INTERFACE I_KeyValueEnumerable EXTENDS __SYSTEM.IQueryInterface

METHOD PUBLIC GetKeyValueEnumerator : I_KeyValueForwardEnumerator
END_METHOD

END_INTERFACE

(* stored: Version 1.1.0.1, ProductVersion 3.1.4024.12
   Itf I_KeyValueEnumerable: Id {b74ab324-78d6-0161-1d05-d267a1cdc16f}
   Method GetKeyValueEnumerator: Id {ddfc352f-fad2-022c-3f33-e1f8a6cd7da1} *)
